// Basic implementation of a default command class for PCS interagtion with internal structure of ``ST_CommandBaseHandshake``.
// Aditional IN and OUT parameters should be declared in the derived implementation.
FUNCTION_BLOCK PUBLIC CommandBase IMPLEMENTS ICommand
VAR_IN_OUT
	(* Use Class Properties for IN_OUT Parameters!!! *)
END_VAR
VAR
	stHandshake		: ST_CommandBaseHandshake;		// Internal variable strukture for communication with PCS.
END_VAR

// OO-Class 
;

// Abort the ``Task`` Execution with the result code ``Cancelled``
METHOD PUBLIC Abort
Done(E_CommandResultCode.Cancelled);
END_METHOD

// Can be used to calculate the ``stHandshake.nProgress`` and ``stHandshake.nSubTask``
METHOD PROTECTED CalculateProgress
IF stHandshake.nResultCode = E_CommandResultCode.Done THEN
	stHandshake.nProgress := 100;
END_IF
END_METHOD

// The method is called in each cycle to execute the funktional part and the states of the command implementation.
METHOD PUBLIC Call
VAR
	bInit		: BOOL;
END_VAR
// Starting Case
stHandshake.bBusy S= bInit := (stHandshake.bExecute AND NOT stHandshake.bBusy);
IF bInit THEN
	stHandshake.nResultCode := E_CommandResultCode.Init;
	Init();
END_IF

// Cancel Case
IF NOT stHandshake.bExecute AND stHandshake.bBusy THEN
	Abort();
END_IF

// Running Case
IF stHandshake.bExecute AND stHandshake.bBusy THEN
	
	// Set Task init on First Call
	stHandshake.nResultCode := E_CommandResultCode.Running;
	IF Task() THEN
		Done(E_CommandResultCode.Done);
	END_IF
		
	CalculateProgress();	
END_IF
END_METHOD

// Can be use to finish the ``Task`` Execution with a ``nResultCode``. 
METHOD PROTECTED Done
VAR_INPUT
	nResultCode		: UINT;
END_VAR
stHandshake.bBusy := stHandshake.bExecute := FALSE;
stHandshake.nResultCode := nResultCode;
END_METHOD

// Will be executed in the same cycle ``stHandshake.bExecute`` changes to ``true``
METHOD PROTECTED Init
VAR_INPUT
END_VAR
stHandshake.nResultCode := E_CommandResultCode.Running;
stHandshake.nProgress := 0;
stHandshake.nSubTask := 0;
END_METHOD

PROPERTY PROTECTED Progress : BYTE
GET
Progress := stHandshake.nProgress;
END_GET
SET
stHandshake.nProgress := Progress;
END_SET
END_PROPERTY

PROPERTY PROTECTED SubTask : UINT
GET
SubTask := stHandshake.nSubTask;
END_GET
SET
stHandshake.nSubTask := SubTask;
END_SET
END_PROPERTY

// Execute the funktional part of the command implementation. Will be executed in the same cycle ``stHandshake.bExecute`` changes to ``true`` after the ``Init`` Method
METHOD PROTECTED Task : BOOL
// Task complete if return true
Task := TRUE;
END_METHOD

END_FUNCTION_BLOCK

(* stored: Version 1.1.0.1, ProductVersion 3.1.4022.7
   POU CommandBase: Id {ada50c45-e2a4-0e1e-2882-6555ee7dd9e0}, SpecialFunc None
   Method Abort: Id {ea835809-8527-04fc-2537-4ead9acb0d0c}
   Method CalculateProgress: Id {a16648df-eb2b-0767-0ec1-b2c892b01c2b}
   Method Call: Id {122b0574-ff69-07fc-29ae-2aea1e238cec}
   Method Done: Id {38ab0c16-9dcb-0710-3b7a-4cc8228c26d9}
   Method Init: Id {73b42678-0303-042f-2b5e-b8719716b1e0}
   Property Progress: Id {11d7213a-75df-05a5-3911-c70fda26068b}
   Get Get: Id {c53dadf5-7315-05cc-3a61-3ca6f99e45f9}
   Set Set: Id {f433abb7-fe0c-0c14-2493-599cdeee1e2b}
   Property SubTask: Id {91ef01b2-b368-094f-0905-247a111f2a9e}
   Get Get: Id {3e9e1d4d-b86f-0b19-192c-a177a58c94f5}
   Set Set: Id {52959122-866e-0ed0-07d0-b14507bb4e0d}
   Method Task: Id {50b60cf9-4807-097f-189d-1bed3be2c16e} *)
